PROGRAM PWM_CTRL
VAR
	
	fbPWM_PROP : FB_PWM;
	
	bOutput_PWM_PROP AT %Q* : BOOL;

END_VAR

// Call the block with a 3-second ramp
fbPWM_PROP(
    fTargetDutyCycle := GVL_THERMAL.fDutyCycle_PROP, nPeriodCycles := 10,
    fRampTime := T#3s, 
    bOut => bOutput_PWM_PROP
);

//probably some PID

END_PROGRAM

(* stored: Version 1.1.0.1
   POU PWM_CTRL: Id {e9a4000a-2bdc-4fc2-aaff-9895c02a3521}, SpecialFunc None *)
